FUNCTION DEGRE2RAD : lreal
VAR_INPUT
	lrAngle : LREAL;
END_VAR
VAR
END_VAR

DEGRE2RAD := lrAngle*PI/180;

END_FUNCTION

(* stored: Version 1.1.0.1, ProductVersion 3.1.4024.11
   POU DEGRE2RAD: Id {1d2279b9-2f42-4930-995a-c27356d14dd3}, SpecialFunc None *)
